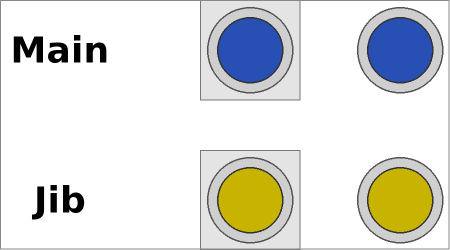
VISUALIZATION VISU_Mode  // 450x250
    Lamp1 (350,150 100x100), variable: GVL.bLampYellow, style: Lamp-Lamp1-Yellow
    Lamp1 (350,0 100x100), variable: GVL.bLampBlue, style: Lamp-Lamp1-Blue
    PushSwitch (200,0 100x100), variable: GVL.bBtnManual, behaviour: TOGGLE, style: Switch-PushSwitch-Blue
    PushSwitch (200,150 100x100), variable: GVL.bBtnAutomatic, behaviour: TOGGLE, style: Switch-PushSwitch-Yellow
    Textfield (0,25 120x50), "Main"
    Textfield (0,175 120x50), "Jib"
END_VISUALIZATION

(* stored: Version 1.1.0.1
   Visu VISU_Mode: Id {f666a14d-cfb3-409f-bc5f-ad3f11df138d} *)
